PROGRAM MAIN
VAR
	fbTimer: FB_TIME;
	fbReceiver: FB_CCS_RECEIVER;
	{attribute 'OPC.UA.DA':='1'}
	drot:			FB_MA_DROT;
	{attribute 'OPC.UA.DA':='1'}
	sim_drot:	FB_SIM_MOTOR;
	
	
	
END_VAR

fbTimer();
fbReceiver(refTimeObj := fbTimer);
//
//Devices
//
drot(sName:='DROT', sMotorName:= 'DrotMotor', 
	 in_lrRotation :=fbReceiver.tracking_ccs.north_angle,
	 in_lrPupil := fbReceiver.tracking_ccs.pupil_angle,
	 in_lrParallactic :=fbReceiver.tracking_ccs.pa,
	 nNOVRAM_DevId:=0);
	 
sim_drot(ptrCfg:=ADR(drot.motor.cfg), ptrStat:=ADR(drot.motor.stat));

END_PROGRAM

(* stored: Version 1.1.0.1, ProductVersion 3.1.4024.11
   POU MAIN: Id {0e8b7f5d-63c1-4068-8341-41a067b6b414}, SpecialFunc None *)
